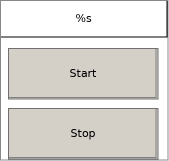
VISUALIZATION Frame_Conveyor  // 169x161
VAR_IN_OUT
	vio_fbConveyor : FB_Conveyor;
END_VAR
    Group (0,0 167x159)
        Button (8,48 150x51), "Start"
            tap vio_fbConveyor.in_bStart
        Button (8,108 150x51), "Stop"
            tap vio_fbConveyor.in_bStop
        Rectangle (0,0 167x37), "%s", text variable: vio_fbConveyor.sModuleName
END_VISUALIZATION

(* stored: Version 1.1.0.1, ProductVersion 3.1.4022.16
   Visu Frame_Conveyor: Id {722a7a19-219e-4eb4-ab3b-4a0dc1e3be14} *)
